FUNCTION_BLOCK FB_1sUPS_BAPI IMPLEMENTS i1sUPS
VAR
	fb1sUps		:FB_S_UPS_BAPI;
END_VAR

PROPERTY bPowerFailDetect : BOOL
GET
bPowerFailDetect:=fb1sUps.bPowerFailDetect;
END_GET
END_PROPERTY

PROPERTY eUpsState : E_S_UPS_State
GET
eUpsState := fb1sUps.eState;
END_GET
END_PROPERTY

METHOD UPSCall
VAR_INPUT
	(*PC AMS Net ID*)
	PcAmsNetId	: AMSNETID;
END_VAR
fb1sUps(sNetID				:=F_CreateAmsNetId(PcAmsNetId),
		iPLCPort			:=_AppInfo.AdsPort,
		tTimeout			:=DEFAULT_ADS_TIMEOUT,
		eUpsMode			:=E_S_UPS_Mode.eSUPS_WrPersistData_Shutdown,
		ePersistentMode		:=E_PersistentMode.SPDM_2PASS,
		tRecoverTime		:=T#10S,
		bPowerFailDetect	=>,
		eState				=>,
		nCapacity			=>,
		bBusy				=>,
		bError				=>,
		nErrID				=>
		);
END_METHOD

END_FUNCTION_BLOCK

(* stored: Version 1.1.0.1, ProductVersion 3.1.4026.12
   POU FB_1sUPS_BAPI: Id {279cc759-b3cd-4952-90bb-d46146b29c9c}, SpecialFunc None
   Property bPowerFailDetect: Id {a89a936d-5a17-4906-9c8d-cec43bd647d4}
   Get Get: Id {c26666b7-54c6-4f24-8c5f-ee8c5c507497}
   Property eUpsState: Id {dad24e9e-cb8b-445c-a7b8-faecd1b5c173}
   Get Get: Id {c5dcc6eb-ab01-4c55-bf5a-60c9fece5ca6}
   Method UPSCall: Id {9f41339e-51b0-4ce2-8c16-04c0d06ce6ec} *)
